Fanuc KAREL source: ks00052.KL

PROGRAM KS00052
%STACKSIZE=65535
%PRIORITY=65535
%NOLOCKGROUP
TYPE
REC_T=STRUCTURE
VALUE : INTEGER
FLAG : BOOLEAN
ENDSTRUCTURE
VAR
A : ARRAY[4] OF REC_T
B : ARRAY[4] OF REC_T
FLAG : BOOLEAN
N : INTEGER
STATUS : INTEGER
PN : STRING[80]
VN : STRING[80]
BEGIN
PN=''
VN='A'
-- UNRESOLVED_PC line 19 opcodes [22 22 1E] marker_code=27
END KS00052
